(* CODESYS project Garage Door.project

Project tree, tasks and I/O mapping:
  Device : CODESYS Control Win V3, 3S - Smart Software Solutions GmbH, order no. 305021, version 3.5.10.40
    application Application
      libraries: Standard, * (System)
      task MainTask (cyclic, interval t#20ms, priority 1) calls PLC_PRG
      program PLC_PRG [LD]
      global variables GVL
      Symbols
*)

// Device/Application/GVL
{attribute 'qualified_only'}
VAR_GLOBAL
	PushButton: BOOL;
	SensorOpen: BOOL;
	SensorClose: BOOL;
	MotorForward: BOOL;
	MotorReverse: BOOL;
	TopLight: BOOL;
END_VAR

// Device/Application/PLC_PRG
PROGRAM PLC_PRG
VAR
	tof01: TOF;
	TON_1: TON;
	Timmer3: TIME;
	TOF_0: TOF;
	Timmer_Elipse_Open_Door: TIME;
	Timmer_MovingDoor_On: TIME;
	Timmer_MovingDoor_off: TIME;
END_VAR

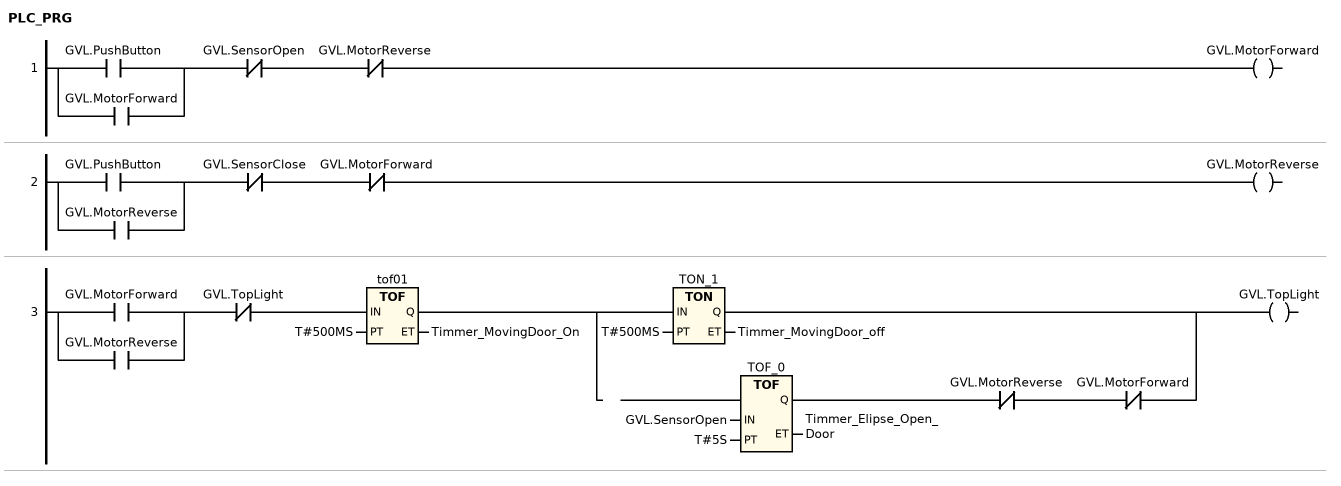
// NETWORK 1
GVL.MotorForward := (GVL.PushButton OR GVL.MotorForward) AND NOT GVL.SensorOpen AND NOT GVL.MotorReverse;

// NETWORK 2
GVL.MotorReverse := (GVL.PushButton OR GVL.MotorReverse) AND NOT GVL.SensorClose AND NOT GVL.MotorForward;

// NETWORK 3
tof01(
    IN := (GVL.MotorForward OR GVL.MotorReverse) AND NOT GVL.TopLight,
    PT := T#500MS,
    ET => Timmer_MovingDoor_On); // TOF
TON_1(IN := tof01.Q, PT := T#500MS, ET => Timmer_MovingDoor_off); // TON
TOF_0(IN := GVL.SensorOpen, PT := T#5S, ET => Timmer_Elipse_Open_Door); // TOF
GVL.TopLight := TON_1.Q OR TOF_0.Q AND NOT GVL.MotorReverse AND NOT GVL.MotorForward;

END_PROGRAM
